// TIA Portal V20 export
DATA_BLOCK "BA010AZCR_UnwinderVirtualAxis"   // DB269, Motion_DB
// stored: InstanceOfName TO_SynchronousAxis, OfSystemLibElement TO_SynchronousAxis, OfSystemLibVersion 9.0
TO_SynchronousAxis   // technology object, version 9.0
// stored: DelayedCoupling Ref BA010AZCR_MasterVirtualAxis, Type TO_SynchronousAxis
   // // inherited from TO_PositioningAxis
   // // inherited from TO_SpeedAxis
   // // inherited from TO_Axis
   // // inherited from TO_Object
   // VAR
   //    VirtualAxis : TO_Struct_VirtualAxis;
   // END_VAR
   // VAR
   //    SynchronizedMotion { S7_SetPoint := 'True'} : TO_Struct_SynchronizedMotion;
   //    StatusSynchronizedMotion { ExternalWritable := 'False'; S7_SetPoint := 'True'} : TO_Struct_StatusSynchronizedMotion;
   // END_VAR
BEGIN
   VirtualAxis.Mode := 1;
   VirtualAxis.Mode := 1;
END_DATA_BLOCK
